// TIA Portal V17 export
// export: Created 2024-06-14T09:52:45.0212781Z, ExportSetting WithDefaults, DisplayName Totally Integrated Automation Portal, DisplayVersion V17, DisplayName TIA Portal Openness, DisplayVersion V17, DisplayName TIA Portal Version Control Interface, DisplayVersion V17, DisplayName Simotion SCOUT TIA, DisplayVersion 5.4.3.0, DisplayName SINAMICS Startdrive Advanced, DisplayVersion V17 SP1 Update 1, DisplayName SINAMICS Startdrive G110M, G120, G120C, G120D, G120P, G115D, DisplayVersion V17 SP1 Update 1, DisplayName SINAMICS Startdrive G130, G150, S120, S150, SINAMICS MV, S210, DisplayVersion V17 SP1 Update 1, DisplayName STEP 7 Professional, DisplayVersion V17, DisplayName STEP 7 Safety, DisplayVersion V17, DisplayName WinCC Professional, DisplayVersion V17
FUNCTION_BLOCK "Enabled_Station"   // FB2, LAD
{ S7_Optimized_Access := 'TRUE' }
VERSION : 0.1
// stored: AutoNumber true, IsIECCheckEnabled false, IsRetainMemResEnabled false, MemoryReserve 100, SetENOAutomatically false, UDAEnableTagReadback false
   VAR_INPUT
      Enable_Station : Bool;
      Enable_Stations : Array[1..6] of Bool;
   END_VAR
   VAR_OUTPUT
      Enabled_Station : Int;
   END_VAR
   VAR
      Station1 : Int;
      Station2 : Int;
      Station3 : Int;
      Station4 : Int;
      Station5 : Int;
      Station6 : Int;
   END_VAR
   VAR_TEMP   // added for the SCL form of the ladder/FBD networks
      _w1 : Bool;
   END_VAR
BEGIN

REGION Network 2: Station-1 Enabled
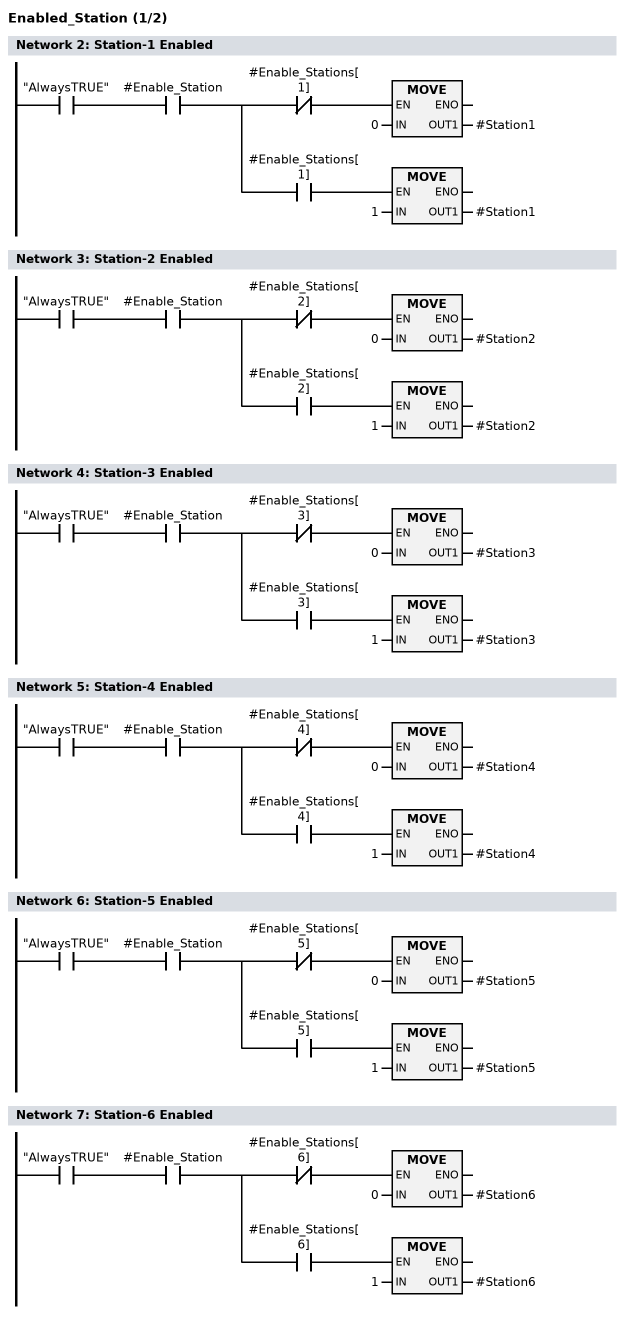
   RUNG wire#powerrail
      Contact( "AlwaysTRUE" )
      Contact( #Enable_Station )
      wire#w1
      I_Contact( #Enable_Stations[1] )
      Move(in := 0, out1 => #Station1)
   END_RUNG
   RUNG wire#w1
      Contact( #Enable_Stations[1] )
      Move(in := 1, out1 => #Station1)
   END_RUNG
   // the same network as SCL:
   #_w1 := "AlwaysTRUE" AND #Enable_Station;
   IF #_w1 AND NOT #Enable_Stations[1] THEN #Station1 := 0; END_IF;
   IF #_w1 AND #Enable_Stations[1] THEN #Station1 := 1; END_IF;
END_REGION

REGION Network 3: Station-2 Enabled
   RUNG wire#powerrail
      Contact( "AlwaysTRUE" )
      Contact( #Enable_Station )
      wire#w1
      I_Contact( #Enable_Stations[2] )
      Move(in := 0, out1 => #Station2)
   END_RUNG
   RUNG wire#w1
      Contact( #Enable_Stations[2] )
      Move(in := 1, out1 => #Station2)
   END_RUNG
   // the same network as SCL:
   #_w1 := "AlwaysTRUE" AND #Enable_Station;
   IF #_w1 AND NOT #Enable_Stations[2] THEN #Station2 := 0; END_IF;
   IF #_w1 AND #Enable_Stations[2] THEN #Station2 := 1; END_IF;
END_REGION

REGION Network 4: Station-3 Enabled
   RUNG wire#powerrail
      Contact( "AlwaysTRUE" )
      Contact( #Enable_Station )
      wire#w1
      I_Contact( #Enable_Stations[3] )
      Move(in := 0, out1 => #Station3)
   END_RUNG
   RUNG wire#w1
      Contact( #Enable_Stations[3] )
      Move(in := 1, out1 => #Station3)
   END_RUNG
   // the same network as SCL:
   #_w1 := "AlwaysTRUE" AND #Enable_Station;
   IF #_w1 AND NOT #Enable_Stations[3] THEN #Station3 := 0; END_IF;
   IF #_w1 AND #Enable_Stations[3] THEN #Station3 := 1; END_IF;
END_REGION

REGION Network 5: Station-4 Enabled
   RUNG wire#powerrail
      Contact( "AlwaysTRUE" )
      Contact( #Enable_Station )
      wire#w1
      I_Contact( #Enable_Stations[4] )
      Move(in := 0, out1 => #Station4)
   END_RUNG
   RUNG wire#w1
      Contact( #Enable_Stations[4] )
      Move(in := 1, out1 => #Station4)
   END_RUNG
   // the same network as SCL:
   #_w1 := "AlwaysTRUE" AND #Enable_Station;
   IF #_w1 AND NOT #Enable_Stations[4] THEN #Station4 := 0; END_IF;
   IF #_w1 AND #Enable_Stations[4] THEN #Station4 := 1; END_IF;
END_REGION

REGION Network 6: Station-5 Enabled
   RUNG wire#powerrail
      Contact( "AlwaysTRUE" )
      Contact( #Enable_Station )
      wire#w1
      I_Contact( #Enable_Stations[5] )
      Move(in := 0, out1 => #Station5)
   END_RUNG
   RUNG wire#w1
      Contact( #Enable_Stations[5] )
      Move(in := 1, out1 => #Station5)
   END_RUNG
   // the same network as SCL:
   #_w1 := "AlwaysTRUE" AND #Enable_Station;
   IF #_w1 AND NOT #Enable_Stations[5] THEN #Station5 := 0; END_IF;
   IF #_w1 AND #Enable_Stations[5] THEN #Station5 := 1; END_IF;
END_REGION

REGION Network 7: Station-6 Enabled
   RUNG wire#powerrail
      Contact( "AlwaysTRUE" )
      Contact( #Enable_Station )
      wire#w1
      I_Contact( #Enable_Stations[6] )
      Move(in := 0, out1 => #Station6)
   END_RUNG
   RUNG wire#w1
      Contact( #Enable_Stations[6] )
      Move(in := 1, out1 => #Station6)
   END_RUNG
   // the same network as SCL:
   #_w1 := "AlwaysTRUE" AND #Enable_Station;
   IF #_w1 AND NOT #Enable_Stations[6] THEN #Station6 := 0; END_IF;
   IF #_w1 AND #Enable_Stations[6] THEN #Station6 := 1; END_IF;
END_REGION

REGION Network 8
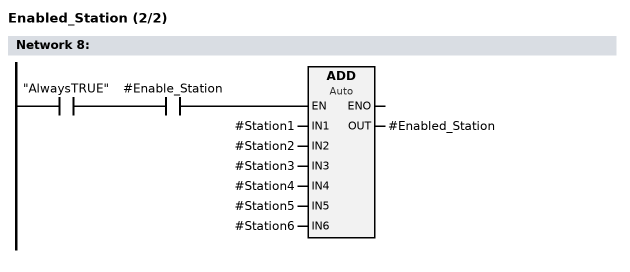
   RUNG wire#powerrail
      Contact( "AlwaysTRUE" )
      Contact( #Enable_Station )
      Add(in1 := #Station1, in2 := #Station2, in3 := #Station3, in4 := #Station4, in5 := #Station5, in6 := #Station6, out => #Enabled_Station)
   END_RUNG
   // the same network as SCL:
   IF "AlwaysTRUE" AND #Enable_Station THEN
       #Enabled_Station := #Station1 + #Station2 + #Station3 + #Station4 + #Station5 + #Station6;
   END_IF;
END_REGION
END_FUNCTION_BLOCK
